KUKA KRL program: wkz4_ok.src, wkz4_ok.dat

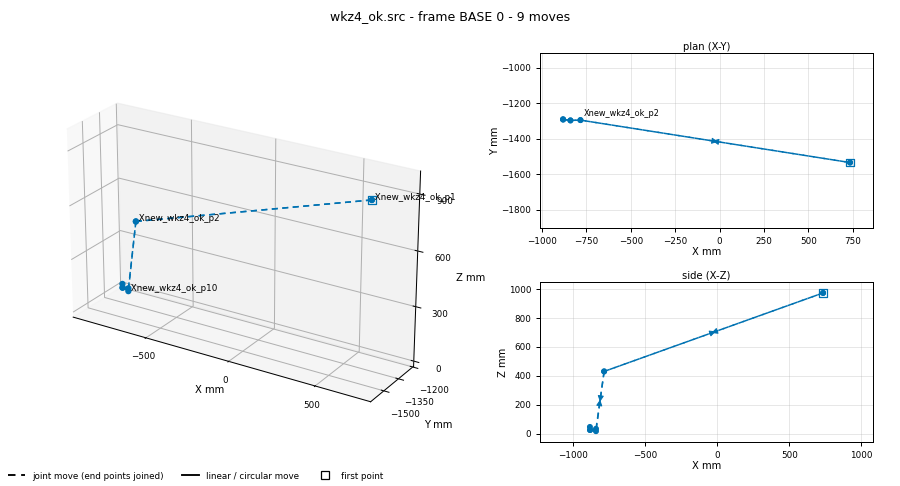
[picture p0: tool path of wkz4_ok.src in frame BASE 0, 9 of 11 moves have a stored position in this frame; points joined in program order, loops and branches not executed]
--- wkz4_ok.src ---
&ACCESS RVP
&REL 5
&COMMENT CHK_TCP_X1
&PARAM DISKPATH = KRC:\R1\Program\TOOL CHANGE
DEF WKZ4_OK ( )

;FOLD INI
  ;FOLD BASISTECH INI
    GLOBAL INTERRUPT DECL 3 WHEN $STOPMESS==TRUE DO IR_STOPM ( )
    INTERRUPT ON 3
    BAS (#INITMOV,0 )
  ;ENDFOLD (BASISTECH INI)
  ;FOLD USER INI
    ;Make your modifications here
  ;ENDFOLD (USER INI)
;ENDFOLD (INI)
;FOLD PTP HOME  Vel= 100 % DEFAULT;%{PE}%V3.2.0,%MKUKATPBASIS,%CMOVE,%VPTP,%P 1:PTP, 2:HOME, 3:, 5:100, 7:DEFAULT
$BWDSTART = FALSE
$H_POS=XHOME
PDAT_ACT=PDEFAULT
BAS (#PTP_DAT )
FDAT_ACT=FHOME
BAS (#FRAMES )
BAS (#VEL_PTP,100 )
PTP  XHOME
;ENDFOLD

; Caracterização dos meios de produção:
; Versão Atual:
; 04/05/2013 12:00 Name: P13.090-R6 CHANGES: Check TCP X1

chk_w4_wechs_ok ( )  ; VERIFICAÇÃO DE FERRAMENTA: GUN X1

;FOLD PTP new_wkz4_ok_p1  Vel=100 % P_OLP1 Tool[4]" " Base[0]  ;%{PE}%R8.3,%MKUKATPBASIS,%CMOVE,%VPTP,%P 1:PTP, 2:new_wkz4_ok_p1, 3:, 5:100, 7:P_OLP1
$BWDSTART = FALSE
PDAT_ACT= PP_OLP1
FDAT_ACT= Fnew_wkz4_ok_p1
BAS(#PTP_PARAMS,100)
PTP Xnew_wkz4_ok_p1
;ENDFOLD
;FOLD PTP new_wkz4_ok_p2  Vel=100 % P_OLP2 Tool[4]" " Base[0]  ;%{PE}%R8.3,%MKUKATPBASIS,%CMOVE,%VPTP,%P 1:PTP, 2:new_wkz4_ok_p2, 3:, 5:100, 7:P_OLP2
$BWDSTART = FALSE
PDAT_ACT= PP_OLP2
FDAT_ACT= Fnew_wkz4_ok_p2
BAS(#PTP_PARAMS,100)
PTP Xnew_wkz4_ok_p2
;ENDFOLD
;FOLD PTP new_wkz4_ok_p10  Vel=100 % P_OLP3 Tool[4]" " Base[0]  ;%{PE}%R8.3,%MKUKATPBASIS,%CMOVE,%VPTP,%P 1:PTP, 2:new_wkz4_ok_p10, 3:, 5:100, 7:P_OLP3
$BWDSTART = FALSE
PDAT_ACT= PP_OLP3
FDAT_ACT= Fnew_wkz4_ok_p10
BAS(#PTP_PARAMS,100)
PTP Xnew_wkz4_ok_p10
;ENDFOLD
;FOLD LIN new_wkz4_ok_p3  Vel=2.00 m/s L_OLP1 Tool[4]" " Base[0] ;%{PE}%R8.3,%MKUKATPBASIS,%CMOVE,%VLIN,%P 1:LIN, 2:new_wkz4_ok_p3, 3:, 5:2.00, 7:L_OLP1
$BWDSTART = FALSE
LDAT_ACT= LL_OLP1
FDAT_ACT= Fnew_wkz4_ok_p3
BAS(#CP_PARAMS,2.00)
LIN Xnew_wkz4_ok_p3
;ENDFOLD
;FOLD LIN new_wkz4_ok_ptcpc  Vel=2.00 m/s L_OLP2 Tool[4]" " Base[0] ;%{PE}%R8.3,%MKUKATPBASIS,%CMOVE,%VLIN,%P 1:LIN, 2:new_wkz4_ok_ptcpc, 3:, 5:2.00, 7:L_OLP2
$BWDSTART = FALSE
LDAT_ACT= LL_OLP2
FDAT_ACT= Fnew_wkz4_ok_ptcpc
BAS(#CP_PARAMS,2.00)
LIN Xnew_wkz4_ok_ptcpc
;ENDFOLD
;FOLD LIN new_wkz4_ok_p4  Vel=2.00 m/s L_OLP3 Tool[4]" " Base[0] ;%{PE}%R8.3,%MKUKATPBASIS,%CMOVE,%VLIN,%P 1:LIN, 2:new_wkz4_ok_p4, 3:, 5:2.00, 7:L_OLP3
$BWDSTART = FALSE
LDAT_ACT= LL_OLP3
FDAT_ACT= Fnew_wkz4_ok_p4
BAS(#CP_PARAMS,2.00)
LIN Xnew_wkz4_ok_p4
;ENDFOLD
;FOLD PTP new_wkz4_ok_p12  Vel=100 % P_OLP4 Tool[4]" " Base[0]  ;%{PE}%R8.3,%MKUKATPBASIS,%CMOVE,%VPTP,%P 1:PTP, 2:new_wkz4_ok_p12, 3:, 5:100, 7:P_OLP4
$BWDSTART = FALSE
PDAT_ACT= PP_OLP4
FDAT_ACT= Fnew_wkz4_ok_p12
BAS(#PTP_PARAMS,100)
PTP Xnew_wkz4_ok_p12
;ENDFOLD
;FOLD PTP new_wkz4_ok_p5  Vel=100 % P_OLP5 Tool[4]" " Base[0]  ;%{PE}%R8.3,%MKUKATPBASIS,%CMOVE,%VPTP,%P 1:PTP, 2:new_wkz4_ok_p5, 3:, 5:100, 7:P_OLP5
$BWDSTART = FALSE
PDAT_ACT= PP_OLP5
FDAT_ACT= Fnew_wkz4_ok_p5
BAS(#PTP_PARAMS,100)
PTP Xnew_wkz4_ok_p5
;ENDFOLD
;FOLD PTP new_wkz4_ok_p6  Vel=100 % P_OLP6 Tool[4]" " Base[0]  ;%{PE}%R8.3,%MKUKATPBASIS,%CMOVE,%VPTP,%P 1:PTP, 2:new_wkz4_ok_p6, 3:, 5:100, 7:P_OLP6
$BWDSTART = FALSE
PDAT_ACT= PP_OLP6
FDAT_ACT= Fnew_wkz4_ok_p6
BAS(#PTP_PARAMS,100)
PTP Xnew_wkz4_ok_p6
;ENDFOLD

;FOLD PTP HOME  Vel= 100 % DEFAULT;%{PE}%V3.2.0,%MKUKATPBASIS,%CMOVE,%VPTP,%P 1:PTP, 2:HOME, 3:, 5:100, 7:DEFAULT
$BWDSTART = FALSE
$H_POS=XHOME
PDAT_ACT=PDEFAULT
BAS (#PTP_DAT )
FDAT_ACT=FHOME
BAS (#FRAMES )
BAS (#VEL_PTP,100 )
PTP  XHOME
;ENDFOLD
END

--- wkz4_ok.dat ---
&ACCESS RVP
&REL 5
&COMMENT CHK_TCP_X1
&PARAM DISKPATH = KRC:\R1\Program\TOOL CHANGE
DEFDAT  wkz4_ok
;FOLD EXTERNAL DECLARATIONS;%{PE}%MKUKATPBASIS,%CEXT,%VCOMMON,%P
;FOLD BASISTECH EXT;%{PE}%MKUKATPBASIS,%CEXT,%VEXT,%P
EXT  BAS (BAS_COMMAND  :IN,REAL  :IN )
DECL INT SUCCESS
;ENDFOLD (BASISTECH EXT)
;FOLD USER EXT;%{E}%MKUKATPUSER,%CEXT,%VEXT,%P
;Make your modifications here
;ENDFOLD (USER EXT)
;ENDFOLD (EXTERNAL DECLARATIONS)

;# ============ START PATH : wkz4_ok =============
DECL FDAT Fnew_wkz4_ok_p1={TOOL_NO 4,BASE_NO 0,IPO_FRAME #BASE,POINT2[] " "}
DECL PDAT PP_OLP1={VEL 100.0,ACC 50.0,APO_DIST 0.0}
DECL E6POS Xnew_wkz4_ok_p1={X 733.906006,Y -1533.59705,Z 974.255981,A 40.8928986,B 72.251297,C -59.2467995,S 2,T 10}
DECL FDAT Fnew_wkz4_ok_p2={TOOL_NO 4,BASE_NO 0,IPO_FRAME #BASE,POINT2[] " "}
DECL PDAT PP_OLP2={VEL 100.0,ACC 50.0,APO_DIST 0.0}
DECL E6POS Xnew_wkz4_ok_p2={X -783.77002,Y -1294.76904,Z 430.299988,A 169.129898,B -0.412400007,C 1.72080004,S 2,T 2}
DECL FDAT Fnew_wkz4_ok_p10={TOOL_NO 4,BASE_NO 0,IPO_FRAME #BASE,POINT2[] " "}
DECL PDAT PP_OLP3={VEL 100.0,ACC 50.0,APO_DIST 0.0}
DECL E6POS Xnew_wkz4_ok_p10={X -840.209778,Y -1296.60596,Z 15.9706802,A 169.129807,B -0.411621988,C 1.72166896,S 18,T 2,E1 0.0,E2 0.0,E3 0.0,E4 0.0,E5 0.0,E6 0.0}
DECL FDAT Fnew_wkz4_ok_p3={TOOL_NO 4,BASE_NO 0,IPO_FRAME #BASE,POINT2[] " "}
DECL E6POS Xnew_wkz4_ok_p3={X -880.810608,Y -1291.45996,Z 24.3598709,A 169.130402,B -0.411863387,C 1.72059906,S 18,T 2,E1 0.0,E2 0.0,E3 0.0,E4 0.0,E5 0.0,E6 0.0}
DECL LDAT LL_OLP1={VEL 2.0,ACC 100.0,APO_DIST 0.0,APO_FAC 0.0,ORI_TYP #VAR,CIRC_TYP #BASE,JERK_FAC 50.0}
DECL FDAT Fnew_wkz4_ok_ptcpc={TOOL_NO 4,BASE_NO 0,IPO_FRAME #BASE,POINT2[] " "}
DECL E6POS Xnew_wkz4_ok_ptcpc={X -882.211609,Y -1290.35803,Z 45.50214,A 169.021698,B -0.529966414,C 0.982510805,S 18,T 2,E1 0.0,E2 0.0,E3 0.0,E4 0.0,E5 0.0,E6 0.0}
DECL LDAT LL_OLP2={VEL 2.0,ACC 100.0,APO_DIST 0.0,APO_FAC 0.0,ORI_TYP #VAR,CIRC_TYP #BASE,JERK_FAC 50.0}
DECL FDAT Fnew_wkz4_ok_p4={TOOL_NO 4,BASE_NO 0,IPO_FRAME #BASE,POINT2[] " "}
DECL E6POS Xnew_wkz4_ok_p4={X -881.683472,Y -1290.75806,Z 23.9873199,A 169.130402,B -0.411851287,C 1.720819,S 18,T 2,E1 0.0,E2 0.0,E3 0.0,E4 0.0,E5 0.0,E6 0.0}
DECL LDAT LL_OLP3={VEL 2.0,ACC 100.0,APO_DIST 0.0,APO_FAC 0.0,ORI_TYP #VAR,CIRC_TYP #BASE,JERK_FAC 50.0}
DECL FDAT Fnew_wkz4_ok_p12={TOOL_NO 4,BASE_NO 0,IPO_FRAME #BASE,POINT2[] " "}
DECL PDAT PP_OLP4={VEL 100.0,ACC 50.0,APO_DIST 0.0}
DECL E6POS Xnew_wkz4_ok_p12={X -839.97998,Y -1296.15198,Z 32.6520004,A 169.129898,B -0.412400007,C 1.72080004,S 2,T 2}
DECL FDAT Fnew_wkz4_ok_p5={TOOL_NO 4,BASE_NO 0,IPO_FRAME #BASE,POINT2[] " "}
DECL PDAT PP_OLP5={VEL 100.0,ACC 50.0,APO_DIST 0.0}
DECL E6POS Xnew_wkz4_ok_p5={X -783.77002,Y -1294.76904,Z 430.299988,A 169.129898,B -0.412400007,C 1.72080004,S 2,T 2}
DECL FDAT Fnew_wkz4_ok_p6={TOOL_NO 4,BASE_NO 0,IPO_FRAME #BASE,POINT2[] " "}
DECL PDAT PP_OLP6={VEL 100.0,ACC 50.0,APO_DIST 0.0}
DECL E6POS Xnew_wkz4_ok_p6={X 733.906006,Y -1533.59705,Z 974.255005,A 40.8931007,B 72.2511978,C -59.2466011,S 2,T 10}
ENDDAT
